PROGRAM FB_TCP400
VAR
END_VAR

// NETWORK 1

END_PROGRAM

(* stored: Version 1.1.0.1, ProductVersion 3.1.4022.3
   POU FB_TCP400: Id {43e95292-7d49-491f-922a-85de6422f5f3}, SpecialFunc None *)
